TEXTLIST TextList_Chauffage
  0 = 'chauffage' | FR: 'CHAUFFAGE' | EN: 'HEATING'
  1 = 'puissance' | FR: 'Puissance' | EN: 'Power'
  2 = 'temp' | FR: 'Température' | EN: 'Temperature'
  3 = 'cons temp' | FR: 'Consigne\ntempérature' | EN: 'Temperature\nsetpoint'
  4 = 'cons puiss' | FR: 'Consigne\npuissance' | EN: 'Power\nsetpoint'
  5 = 'cons temp' | FR: 'Consigne temp.' | EN: 'Temp. setpoint'
  6 = 'maintien' | FR: 'Durée de maintien' | EN: 'Hold time'
  7 = 'delta' | FR: 'Variation de temp.' | EN: 'Temp. variation'
  8 = 'max stab' | FR: 'Durée max. de stabilisation' | EN: 'Max. stabilization time'
  9 = 'cons temp' | FR: 'Consigne température' | EN: 'Temperature setpoint'
  10 = 'delta' | FR: 'Variation de température' | EN: 'Temperature variation'
  11 = 'puissance bords' | FR: 'Puissance bords' | EN: 'Borders power'
  12 = 'Tc Ctrl' | FR: 'Thermocouples de régulation' | EN: 'Regulation thermocouples'
  13 = 'Tc Disp' | FR: 'Thermocouples de sécurité' | EN: 'Security thermocouples'
   = ''
END_TEXTLIST

(* stored: Version 1.1.0.1, ProductVersion 3.1.4024.10
   TextList TextList_Chauffage: Id {c932722d-81af-4fb1-be90-aea2e1a8088b} *)
